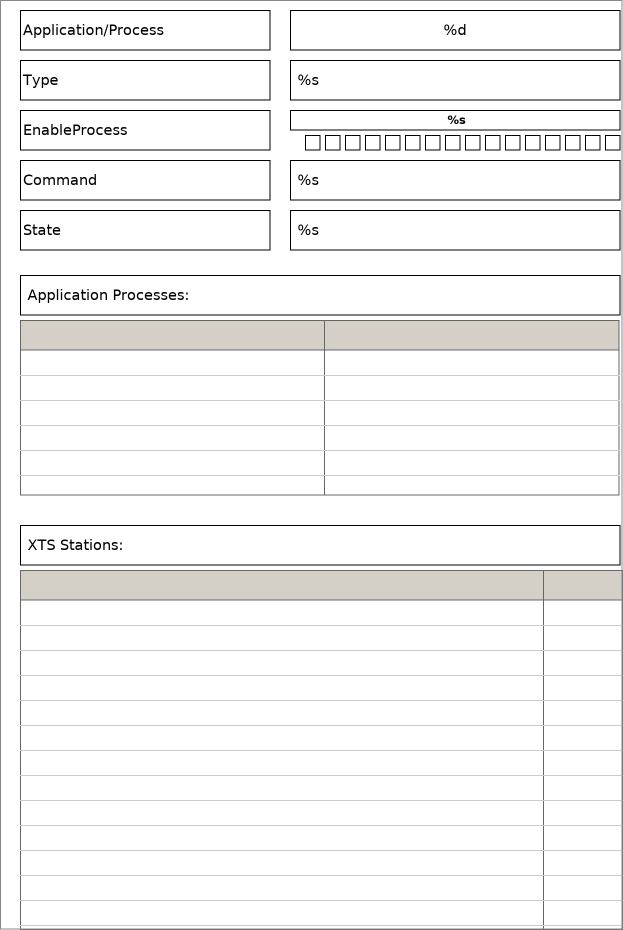
VISUALIZATION T_PROCESS_VISU  // 623x930
VAR_IN_OUT
	nSelectedProcess    : UINT; // selected process index
  EnableProcess       : ARRAY[1..GVL_PROCESS.MAX_PROCESS] OF WORD;
  ProcessCmd          : ARRAY[1..GVL_PROCESS.MAX_PROCESS] OF E_STATION_CTRL;
  ProcessState        : ARRAY[1..GVL_PROCESS.MAX_PROCESS] OF E_STATION_STATE;
  StationState        : ARRAY[1..MAX_STATION] OF ST_STATION_STATE;
  bStationEnabled     : ARRAY[1..MAX_STATION] OF BOOL;
END_VAR
    Rectangle (20,10 250x40), "Application/Process"
    Rectangle (290,10 330x40), "%d", text variable: nSelectedProcess
        OnMouseClick: write the text variable via VisuDialogs.Numpad, min 1, max GVL_PROCESS.MAX_PROCESS, title 'Selected Process'
    Rectangle (20,160 250x40), "Command"
    Rectangle (20,210 250x40), "State"
    Rectangle (20,60 250x40), "Type"
    Rectangle (20,110 250x40), "EnableProcess"
    Rectangle (290,60 330x40), "%s", text variable: GVL_PROCESS.Process[nSelectedProcess]._eType
    Rectangle (290,160 330x40), "%s", text variable: GVL_PROCESS.Process[nSelectedProcess]._eProcessCmd
    Rectangle (290,210 330x40), "%s", text variable: GVL_PROCESS.Process[nSelectedProcess]._eProcessState
    Rectangle (290,110 330x20), "%s", text variable: MAIN.sProcessEnableMask
    Rectangle (605,135 15x15)
        toggle EnableProcess[nSelectedProcess].0
    Rectangle (585,135 15x15)
        toggle EnableProcess[nSelectedProcess].1
    Rectangle (565,135 15x15)
        toggle EnableProcess[nSelectedProcess].2
    Rectangle (545,135 15x15)
        toggle EnableProcess[nSelectedProcess].3
    Rectangle (525,135 15x15)
        toggle EnableProcess[nSelectedProcess].4
    Rectangle (505,135 15x15)
        toggle EnableProcess[nSelectedProcess].5
    Rectangle (485,135 15x15)
        toggle EnableProcess[nSelectedProcess].6
    Rectangle (465,135 15x15)
        toggle EnableProcess[nSelectedProcess].7
    Table (20,570 540x360), data array: StationState
        p3854506369: StationState[INDEX].eState
        p1892666644: StationState[INDEX].nMask
        p338671338: StationState[INDEX].nMoverId
        p2170511999: StationState[INDEX].nQueue
    Table (543,570 80x360), data array: bStationEnabled
        p3854506369: bStationEnabled[INDEX]
    Rectangle (445,135 15x15)
        toggle EnableProcess[nSelectedProcess].8
    Rectangle (425,135 15x15)
        toggle EnableProcess[nSelectedProcess].9
    Rectangle (405,135 15x15)
        toggle EnableProcess[nSelectedProcess].10
    Rectangle (385,135 15x15)
        toggle EnableProcess[nSelectedProcess].11
    Rectangle (365,135 15x15)
        toggle EnableProcess[nSelectedProcess].12
    Rectangle (345,135 15x15)
        toggle EnableProcess[nSelectedProcess].13
    Rectangle (325,135 15x15)
        toggle EnableProcess[nSelectedProcess].14
    Rectangle (305,135 15x15)
        toggle EnableProcess[nSelectedProcess].15
    Rectangle (20,525 600x40), "XTS Stations:"
    Rectangle (20,275 600x40), "Application Processes:"
    Table (20,320 329x175), data array: ProcessState
        p3854506369: ProcessState[INDEX]
    Table (324,320 295x175), data array: ProcessCmd
        p3854506369: ProcessCmd[INDEX]
END_VISUALIZATION

(* stored: Version 1.1.0.1, ProductVersion 3.1.4024.12
   Visu T_PROCESS_VISU: Id {a84a32b9-fc42-4371-8f15-ddb905c75252} *)
